// Mitsubishi GX Works2 project: 실린더응용4   PLC: Q02/Q02H

PROGRAM MAIN
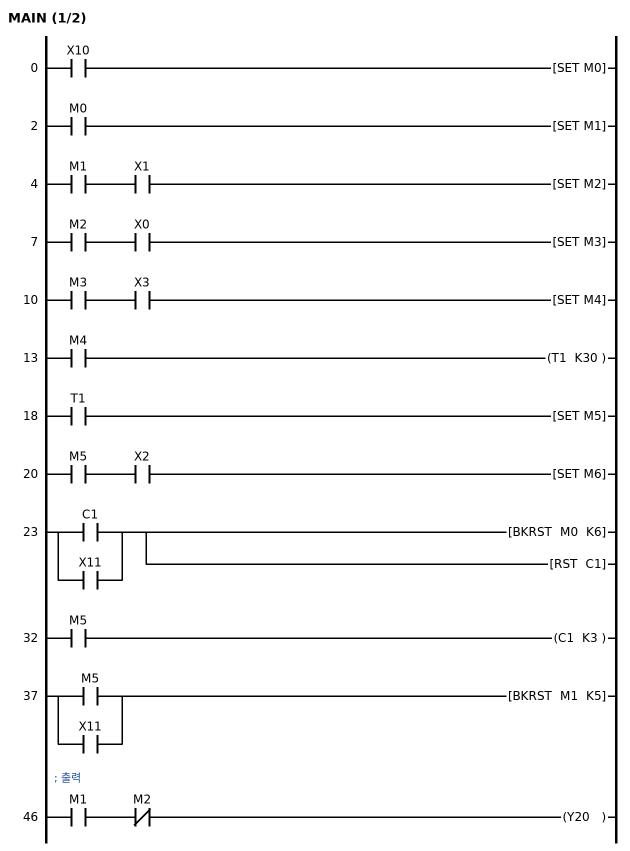
0     LD      X10
      SET     M0
2     LD      M0
      SET     M1
4     LD      M1
      AND     X1
      SET     M2
7     LD      M2
      AND     X0
      SET     M3
10    LD      M3
      AND     X3
      SET     M4
13    LD      M4
      OUT     T1 K30
18    LD      T1
      SET     M5
20    LD      M5
      AND     X2
      SET     M6
23    LD      C1
      OR      X11
      BKRST   M0 K6
      RST     C1
32    LD      M5
      OUT     C1 K3
37    LD      M5
      OR      X11
      BKRST   M1 K5
; 출력
46    LD      M1
      ANI     M2
      OUT     Y20
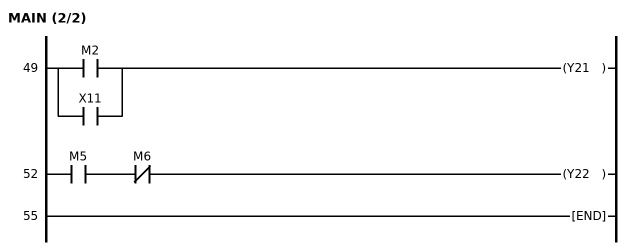
49    LD      M2
      OR      X11
      OUT     Y21
52    LD      M5
      ANI     M6
      OUT     Y22
55    END
END_PROGRAM
